// Type ANY in struct format extended with value of type STRING(255)
TYPE T_Generic_Ex : ST_GENERIC; END_TYPE

(* stored: Version 1.1.0.1, ProductVersion 3.1.4024.4
   DUT T_Generic_Ex: Id {aa5d3600-3cb5-485d-8937-65a2f746eac5} *)
